TYPE csp_case_feed_magazine_accU_osDepth_enum :
(
	CSP_CASE_FEED_MAGAZINE_ACCU_OSDEPTH_STATUS_NOT_INITIALIZED 									:= 0,
	CSP_CASE_FEED_MAGAZINE_ACCU_OSDEPTH_STATUS_DISABLED 										:= 10,
	CSP_CASE_FEED_MAGAZINE_ACCU_OSDEPTH_STATUS_POSITION_CHECK									:= 20,
	CSP_CASE_FEED_MAGAZINE_ACCU_OSDEPTH_STATUS_ENABLE_REQUEST 									:= 30,
	CSP_CASE_FEED_MAGAZINE_ACCU_OSDEPTH_STATUS_ENABLED 											:= 40,
	CSP_CASE_FEED_MAGAZINE_ACCU_OSDEPTH_STATUS_ABS_MOVE_REQUEST									:= 50,
	CSP_CASE_FEED_MAGAZINE_ACCU_OSDEPTH_STATUS_ABS_MOVING										:= 60,
	CSP_CASE_FEED_MAGAZINE_ACCU_OSDEPTH_STATUS_STOP_REQUEST 									:= 70,
	CSP_CASE_FEED_MAGAZINE_ACCU_OSDEPTH_STATUS_DISABLE_REQUEST 									:= 80,
	CSP_CASE_FEED_MAGAZINE_ACCU_OSDEPTH_STATUS_DISABLING 										:= 90
) := CSP_CASE_FEED_MAGAZINE_ACCU_OSDEPTH_STATUS_NOT_INITIALIZED;
END_TYPE

(* stored: Version 1.1.0.1, ProductVersion 3.1.4022.18
   DUT csp_case_feed_magazine_accU_osDepth_enum: Id {d85d7bac-072a-4ec1-912d-86b6fe2df9cd} *)
